// TIA Portal V21 export
VAR_GLOBAL   // PLC tag table "Default tag table"
   Start AT %I0.0 : Bool;   // Start Button
   AutoON AT %I0.1 : Bool;   // Process Running
   Stop AT %I0.2 : Bool;   // Stop Button
   EmgStop AT %I0.3 : Bool;   // Emergency Stop
   Valve AT %Q1.0 : Bool;   // Control Valve
END_VAR
